{attribute 'reflection'}
FUNCTION_BLOCK PUBLIC FB_DevDigitalOutput EXTENDS FB_DevBase
VAR_INPUT
	bCmdOn			: BOOL ; // command output status
END_VAR
VAR_OUTPUT
	bOutputState	: BOOL := FALSE ; // State of physical output
END_VAR
VAR
	qbOutput AT%Q* : BOOL ; // Output to physical device
END_VAR

// Call base function
SUPER^(refFbFault := refFbFault);


// Call private functions
ExecSetOutput();
ExecSetFeedback();

METHOD PRIVATE ExecSetFeedback : BOOL
VAR_INPUT
END_VAR
// Set feedback 
bOutputState := qbOutput ;
END_METHOD

METHOD PRIVATE ExecSetOutput : BOOL
VAR_INPUT
END_VAR
// Set Output to physical device
IF bSafetyOk AND (bEnable OR bCmdManual) THEN 
	qbOutput := bCmdOn ; 
ELSE 
	qbOutput S= FALSE ; 
END_IF
END_METHOD

METHOD PUBLIC Init : BOOL
VAR_INPUT
	// Location data for messages  
	nId			: UDINT ; // Identification number of object
	nParentId	: UDINT ; // Id of higher level If aplicable (0 = no parent)
END_VAR
// ====== Set init to true =====
	bInitOk	:= TRUE ; 

// ====== Calculate device id =====
	bInitOk :=	ExecIdentifyDevice(nId,nParentId, E_ComponentTypes.DiOutput) AND bInitOk;

// ====== Set feedback =====
	Init := bInitOk;
END_METHOD

END_FUNCTION_BLOCK

(* stored: Version 1.1.0.1, ProductVersion 3.1.4024.10
   POU FB_DevDigitalOutput: Id {88d6c6d5-b226-0e14-13a4-cf37841a6f20}, SpecialFunc None
   Folder Private: Id {42798e24-c83a-0025-1549-bf054f87d68b}
   Method ExecSetFeedback: Id {088b4f01-a991-060d-3dfa-d513c0f36526}
   Method ExecSetOutput: Id {8f3954a4-6490-0db9-292c-4d4bf3f054ec}
   Method Init: Id {ef1011e1-65a5-0950-2f24-8f4c79c4e032} *)
